Staubli VAL3: disableQueue.pgx

public program disableQueue(num x_nConvNum (dimensions=1))
begin
  // When this program is called, the queuing of detected objects is
  //  suspended until the program enableQueue() is called. But you must
  //  call the program flushQueue() before enableQueue() to flush the
  //  queue.
  //
  // Input Param
  //  x_nConvNum : Conveyor number
  //
  // Output param
  //  none       :
  //
  //----------------------------------------------------------------
  //
  switch x_nConvNum
    case 0
      call cnv0:disableQueue()
    break
    case 1
      call cnv1:disableQueue()
    break
  endSwitch
end
